// A re-run re-executes the registered set; it does not redefine it. Reset clears

// the verdict and the counts, and keeps the label, the location and the budgets

// the test claimed at registration.
FUNCTION_BLOCK TEST_JournalResetKeepsWhatWasRegistered IMPLEMENTS I_Test
VAR
	Subject		   : TestJournal;
	Handle		   : TestVerdict;
	Budgets		   : ST_TestBudgets;
	Got			   : ST_TestBudgets;
	ExpectedCycles : UDINT;
	ActualCycles   : UDINT;
	ExpectedCount  : UDINT;
	ActualCount	   : UDINT;
END_VAR

METHOD Run : BOOL
VAR_INPUT
	Enable : BOOL;
	Test   : I_TestAssertions;
END_VAR
Budgets.Body.Cycles		 := 11;
Budgets.Body.IsCyclesSet := TRUE;
Subject.SetBudgets(Budgets);
Handle.Target(Subject);
Subject.Begin('first run', 'Verifier.Somewhere');
Handle.Fail('deliberate');
Subject.Finish(E_TestStatus.Passed);
Handle.Untarget();
Test.AssertTrue(Subject.Status = E_TestStatus.Failed, 'failed on the first run');
Subject.Reset();
Test.AssertTrue(Subject.Status = E_TestStatus.NotStarted, 'verdict cleared');
Test.AssertTrue(Subject.Kind = E_FailureKind.None, 'failure kind cleared');
ExpectedCount := 0;
ActualCount	  := Subject.AssertionCount;
Test.AssertEqual(ExpectedCount, ActualCount, 'checks cleared');
Got			   := Subject.Budgets;
ExpectedCycles := 11;
ActualCycles   := Got.Body.Cycles;
Test.AssertEqual(ExpectedCycles, ActualCycles, 'the claimed budget survived the reset');
Run := TRUE;
END_METHOD

END_FUNCTION_BLOCK

(* stored: Version 1.1.0.1, ProductVersion 3.1.4026.18
   POU TEST_JournalResetKeepsWhatWasRegistered: Id {0c7cfbbe-b6d1-442b-9e14-509acdd236bf}, SpecialFunc None
   Folder I_Test: Id {5123b4d0-a268-4000-8cdf-e8f27934ed2d}
   Method Run: Id {1aaab87a-51f2-4b30-8358-18e076521554} *)
